TEXTLIST TL_SingleAxisJogMode_1
  0 = 'Standard slow'
  1 = 'Standard fast'
  2 = 'Continous'
  3 = 'Inching'
  4 = 'Inching modulo'
   = ''
END_TEXTLIST

(* stored: Version 1.1.0.1, ProductVersion 3.1.4024.12
   TextList TL_SingleAxisJogMode_1: Id {611b2ecb-97f4-410f-99c6-68cb261cd800} *)
